// TIA Portal V20 export
VAR_GLOBAL   // PLC tag table "BarcodeReader_DP2"
   "DP2-TriggerEnable" AT %Q152.0 : Bool;
   "DP2-Trigger" AT %Q152.1 : Bool;
   "DP2-TriggerReady" AT %I164.0 : Bool;
   "DP2-TriggerAck" AT %I164.1 : Bool;
   "DP2-Acquiring" AT %I164.2 : Bool;
   "DP2-MissedAcq" AT %I164.3 : Bool;
   "DP2-TriggerID" AT %IW165 : Word;
   "DP2-BufferResultsEnable" AT %Q153.0 : Bool;
   "DP2-ResultsAck" AT %Q153.1 : Bool;
   "DP2-Decoding" AT %I167.0 : Bool;
   "DP2-Decode Complete" AT %I167.1 : Bool;
   "DP2-Results Buffer Overrun" AT %I167.2 : Bool;
   "DP2-Results Available" AT %I167.3 : Bool;
   "DP2-General Fault" AT %I167.7 : Bool;
   "DP2-Train Code" AT %Q154.0 : Bool;
   "DP2-Train Match String" AT %Q154.1 : Bool;
   "DP2-Train Focus" AT %Q154.2 : Bool;
   "DP2-Train Brightness" AT %Q154.3 : Bool;
   "DP2-Untrain" AT %Q154.4 : Bool;
   "DP2-Execute DMCC" AT %Q154.6 : Bool;
   "DP2-Set Match String" AT %Q154.7 : Bool;
   "DP2-Train Code Ack" AT %I168.0 : Bool;
   "DP2-Train Match String Ack" AT %I168.1 : Bool;
   "DP2-Train Focus Ack" AT %I168.2 : Bool;
   "DP2-Train Brightness Ack" AT %I168.3 : Bool;
   "DP2-Untrain Ack" AT %I168.4 : Bool;
   "DP2-Execute DMCC Ack" AT %I168.6 : Bool;
   "DP2-Set Match String Ack" AT %I168.7 : Bool;
   "DP2-UserData Option" AT %QW155 : Word;
   "DP2-UserData Length" AT %QW157 : Word;
   "DP2-UserData[0]" AT %QB159 : Byte;
   "DP2-UserData[1]" AT %QB160 : Byte;
   "DP2-UserData[2]" AT %QB161 : Byte;
   "DP2-UserData[3]" AT %QB162 : Byte;
   "DP2-UserData[4]" AT %QB163 : Byte;
   "DP2-UserData[5]" AT %QB164 : Byte;
   "DP2-UserData[6]" AT %QB165 : Byte;
   "DP2-UserData[7]" AT %QB166 : Byte;
   "DP2-UserData[8]" AT %QB167 : Byte;
   "DP2-UserData[9]" AT %QB168 : Byte;
   "DP2-UserData[10]" AT %QB169 : Byte;
   "DP2-UserData[11]" AT %QB170 : Byte;
   "DP2-UserData[12]" AT %QB171 : Byte;
   "DP2-UserData[13]" AT %QB172 : Byte;
   "DP2-UserData[14]" AT %QB173 : Byte;
   "DP2-UserData[15]" AT %QB174 : Byte;
   "DP2-ResultID" AT %IW169 : Word;
   "DP2-Result Code" AT %IW172 : Word;
   "DP2-Read / No Read" AT %I172.0 : Bool;
   "DP2-Validated / Not Validated" AT %I172.1 : Bool;
   "DP2-Verified / Not Verified" AT %I172.2 : Bool;
   "DP2-Acquisition Trigger Overrun" AT %I172.3 : Bool;
   "DP2-Acquisition Buffer Overflow" AT %I172.4 : Bool;
   "DP2-Result Extended" AT %IW173 : Word;
   "DP2-Result Length" AT %IW175 : Word;
   "DP2-InspectionResults[0]" AT %IB177 : Byte;
   "DP2-InspectionResults[1]" AT %IB178 : Byte;
   "DP2-InspectionResults[2]" AT %IB179 : Byte;
   "DP2-InspectionResults[3]" AT %IB180 : Byte;
   "DP2-InspectionResults[4]" AT %IB181 : Byte;
   "DP2-InspectionResults[5]" AT %IB182 : Byte;
   "DP2-InspectionResults[6]" AT %IB183 : Byte;
   "DP2-InspectionResults[7]" AT %IB184 : Byte;
   "DP2-InspectionResults[8]" AT %IB185 : Byte;
   "DP2-InspectionResults[9]" AT %IB186 : Byte;
   "DP2-InspectionResults[10]" AT %IB187 : Byte;
   "DP2-InspectionResults[11]" AT %IB188 : Byte;
   "DP2-InspectionResults[12]" AT %IB189 : Byte;
   "DP2-InspectionResults[13]" AT %IB190 : Byte;
   "DP2-InspectionResults[14]" AT %IB191 : Byte;
   "DP2-InspectionResults[15]" AT %IB192 : Byte;
   "Result data_DP2" AT %I177.0 : "Global.BarCode";
   UserData_DP2 AT %Q159.0 : "Global.BarCode";
   ContinousGetResults_DP2 AT %M210.1 : Bool;
   TrainFocus_DP2 AT %M210.2 : Bool;
END_VAR
